Yaskawa INFORM job: 01-SAFETY.JBI

/JOB
//NAME 01-SAFETY
///FOLDERNAME OTHER
//POS
///NPOS 1,1,0,0,0,0
///TOOL 0
///POSTYPE ROBOT
///RECTAN
///RCONF 0,0,1,0,0,0,0,0,0,0,0,0,0,0,0,0,0,0,0,0,0,0,0,0
C00000=1690.060,1.247,150.034,-0.1579,-76.2645,0.1527
///RCONF 0,0,0,0,0,0,0,0,0,0,0,0,0,0,0,0,0,0,0,0,0,0,0,0
BC00000=0.020
//INST
///DATE 2024/02/28 12:58
///ATTR SC,RW,RJ
////FRAME ROBOT
///GROUP1 RB1,BS1
NOP
*START
MOVJ C00000 BC00000 VJ=20.00
JUMP *START
END
